FUNCTION F_UpdateFunc : REAL
VAR_INPUT
	bUpdateValue : BOOL;
	fNewValue : REAL; 
	stMotorParameter : ST_MotorParams; 
END_VAR
VAR
END_VAR

IF bUpdateValue THEN
	stMotorParameter.fMaxSpeed := fNewValue; 
	ELSE
		stMotorParameter.fMaxSpeed := stMotorParameter.fMaxSpeed; 

END_IF;

END_FUNCTION

(* stored: Version 1.1.0.1, ProductVersion 3.1.4024.12
   POU F_UpdateFunc: Id {58692343-0c85-4974-b460-9cdebb0d89ec}, SpecialFunc None *)
